(* IEC 61131-3 sources: SysmacStudiohelper-skill/assets, 2 files *)

(* ---- FB_Cylinder2Coil.iec ---- *)
FUNCTION_BLOCK FB_Cylinder2Coil
VAR_INPUT
    Enable : BOOL;
    Reset : BOOL;
    CmdHome : BOOL;
    CmdWork : BOOL;
    PermitHome : BOOL;
    PermitWork : BOOL;
    HomeSensor : BOOL;
    WorkSensor : BOOL;
    CycleMs : UDINT;
    TimeoutMs : UDINT;
END_VAR
VAR_OUTPUT
    HomeValve : BOOL;
    WorkValve : BOOL;
    AtHome : BOOL;
    AtWork : BOOL;
    Busy : BOOL;
    Fault : BOOL;
    FaultID : UINT;
END_VAR
VAR
    Elapsed : UDINT;
    PreviousHome : BOOL;
    PreviousWork : BOOL;
END_VAR
//{st}
(* Device function only: no conveyor, material sensor or machine step number.
   CycleMs must match one invocation per task cycle. Parameters are caller-owned.
   De-energizing a bistable valve does not imply mechanical stopping/retraction. *)
AtHome := HomeSensor AND NOT WorkSensor;
AtWork := WorkSensor AND NOT HomeSensor;
IF Reset AND NOT CmdHome AND NOT CmdWork AND NOT (HomeSensor AND WorkSensor) THEN
    Fault := FALSE; FaultID := 0;
END_IF;
IF Enable THEN
    IF (CycleMs = 0) OR (TimeoutMs = 0) OR (CycleMs > TimeoutMs) THEN
        Fault := TRUE; FaultID := 1;
    ELSIF HomeSensor AND WorkSensor THEN
        Fault := TRUE; FaultID := 2;
    ELSIF CmdHome AND CmdWork THEN
        Fault := TRUE; FaultID := 3;
    END_IF;
END_IF;
HomeValve := Enable AND NOT Fault AND CmdHome AND PermitHome AND NOT CmdWork;
WorkValve := Enable AND NOT Fault AND CmdWork AND PermitWork AND NOT CmdHome;
Busy := (HomeValve AND NOT AtHome) OR (WorkValve AND NOT AtWork);
IF (HomeValve <> PreviousHome) OR (WorkValve <> PreviousWork) OR NOT Busy THEN
    Elapsed := 0;
ELSIF Elapsed >= TimeoutMs THEN
    Fault := TRUE; FaultID := 4;
ELSIF CycleMs >= TimeoutMs - Elapsed THEN
    Elapsed := TimeoutMs;
ELSE Elapsed := Elapsed + CycleMs;
END_IF;
PreviousHome := HomeValve; PreviousWork := WorkValve;
IF Fault THEN HomeValve := FALSE; WorkValve := FALSE; Busy := FALSE; END_IF;
//{end}
END_FUNCTION_BLOCK

(* ---- PRG_Sequence.st ---- *)
(* Program-section fragment, not a full importable project.
   Locals: Step : UINT; Cyl01 : FB_Cylinder2Coil;
   Required caller/global BOOLs: Enable, Reset, StartNewPart, DestinationSensor,
   HomeSensor, WorkSensor, PermitHome, PermitWork, BeltRun, HomeValve, WorkValve.
   UDINTs: TaskCycleMs, CylinderTimeoutMs. All physical mapping is project-owned.
   Example cycle: feed, extend, retract, await next part.
   StartNewPart must be the template's rearmed new-part event, not a held sensor.
   Transitional Step lives HERE, not inside the cylinder FB. *)
IF NOT Enable THEN
    Step := 0;
ELSIF Reset AND ((Step = 0) OR (Step = 900)) AND HomeSensor AND NOT WorkSensor AND NOT DestinationSensor AND NOT Cyl01.Fault THEN
    Step := 10;
ELSIF Cyl01.Fault THEN
    Step := 900;
ELSE
    CASE Step OF
        10: IF StartNewPart THEN Step := 20; END_IF;
        20: IF DestinationSensor THEN Step := 30; END_IF;
        30: IF WorkSensor AND NOT HomeSensor THEN Step := 40; END_IF;
        40: IF HomeSensor AND NOT WorkSensor THEN Step := 10; END_IF;
        0, 900: ;
        ELSE Step := 900;
    END_CASE;
END_IF;
(* Compute commands AFTER transitions: arrival stops belt and requests Work now. *)
BeltRun := Enable AND (Step = 20) AND NOT Cyl01.Fault;
Cyl01(Enable := Enable, Reset := Reset,
    CmdWork := (Step = 30), CmdHome := (Step = 40),
    PermitWork := PermitWork, PermitHome := PermitHome,
    HomeSensor := HomeSensor, WorkSensor := WorkSensor,
    CycleMs := TaskCycleMs, TimeoutMs := CylinderTimeoutMs,
    HomeValve => HomeValve, WorkValve => WorkValve);
IF Cyl01.Fault THEN BeltRun := FALSE; Step := 900; END_IF;
